FUNCTION_BLOCK FB_Ampelstatus
VAR_INPUT
	eState : eBetriebszustand;
END_VAR
VAR_OUTPUT
	bLightRed : BOOL;
	bLightYellow : BOOL;
	bLightGreen : BOOL;
END_VAR
VAR
	fbBlinkRed : FB_Blinklicht;
	fbBlinkYellow : FB_Blinklicht;
	fbBlinkGreen : FB_Blinklicht;
END_VAR

fbBlinkRed(bEinAus:= , tPeriode:= T#2S, bBlink=> bLightRed);
fbBlinkYellow(bEinAus:= , tPeriode:= T#2S, bBlink=> bLightYellow);
fbBlinkGreen(bEinAus:= , tPeriode:= T#2S, bBlink=> bLightGreen);

CASE eState OF
	0: //WARNING, Nicht fehlerbehafteter/ungeplanter Stop
	fbBlinkRed.bEinAus := FALSE;
	fbBlinkYellow.bEinAus := TRUE;
	fbBlinkGreen.bEinAus := FALSE;

	1: //ERROR, Fehlerbehafteter Stop
	fbBlinkRed.bEinAus := TRUE;
	fbBlinkYellow.bEinAus := FALSE;
	fbBlinkGreen.bEinAus := FALSE;

	2: //STOP, Geplanter Stop
	fbBlinkRed.bEinAus := TRUE;
	fbBlinkYellow.bEinAus := TRUE;
	fbBlinkGreen.bEinAus := FALSE;
	
	3: //OFF, Nicht Betriebsbereit
	fbBlinkRed.bEinAus := FALSE;
	fbBlinkYellow.bEinAus := FALSE;
	fbBlinkGreen.bEinAus := FALSE;
	bLightRed := TRUE;
	bLightYellow := FALSE;
	bLightGreen := FALSE;
	
	4: //INIT, Herstellung betriebsbereit
	fbBlinkRed.bEinAus := FALSE;
	fbBlinkYellow.bEinAus := FALSE;
	fbBlinkGreen.bEinAus := TRUE;
	
	5: //PROD, Betrieb
	fbBlinkRed.bEinAus := FALSE;
	fbBlinkYellow.bEinAus := FALSE;
	fbBlinkGreen.bEinAus := FALSE;
	bLightRed := FALSE;
	bLightYellow := FALSE;
	bLightGreen := TRUE;
		
	6: //READY, Betriebsbereit
	fbBlinkRed.bEinAus := FALSE;
	fbBlinkYellow.bEinAus := TRUE;
	fbBlinkGreen.bEinAus := TRUE;
	
	7: //DONE, Betrieb abgeschlosen
	fbBlinkRed.bEinAus := FALSE;
	fbBlinkYellow.bEinAus := FALSE;
	fbBlinkGreen.bEinAus := FALSE;
	bLightRed := FALSE;
	bLightYellow := TRUE;
	bLightGreen := TRUE;
	
	8: //SETUP, Wartung
	fbBlinkRed.bEinAus := FALSE;
	fbBlinkYellow.bEinAus := FALSE;
	fbBlinkGreen.bEinAus := FALSE;
	bLightRed := FALSE;
	bLightYellow := TRUE;
	bLightGreen := FALSE;
	
END_CASE

END_FUNCTION_BLOCK

(* stored: Version 1.1.0.1, ProductVersion 3.1.4024.15
   POU FB_Ampelstatus: Id {98d0a674-dfea-4554-a87b-f1a228891480}, SpecialFunc None *)
